FUNCTION_BLOCK Hexapod_Leg
VAR_INPUT
	Axis1, Axis2, Axis3	: Axis;
END_VAR
VAR_OUTPUT
END_VAR
VAR
	Axis_Leg		: ARRAY [1..3] OF Axis;
	Axis_Number		: INT;
	Axis_HomeDone	: ARRAY [1..3] OF BOOL;
	HomeDone		: BOOL;
END_VAR

Axis_Leg[1] := Axis1;
Axis_Leg[2] := Axis2;
Axis_Leg[3] := Axis3;

METHOD Home
VAR_INPUT
	Axis1_HomeSet	: BOOL;
	Axis2_HomeSet	: BOOL;
	Axis3_HomeSet	: BOOL;
END_VAR
VAR_OUTPUT	
END_VAR
VAR
	Axis_HomeSet	: BOOL;
END_VAR
IF Axis_HomeDone[1] AND Axis_HomeDone[2] AND Axis_HomeDone[2] THEN
	HomeDone := TRUE;
END_IF

Axis_HomeDone[1] := Axis1.State_HomeDone;
Axis_HomeDone[2] := Axis2.State_HomeDone;
Axis_HomeDone[3] := Axis3.State_HomeDone;
END_METHOD

PROPERTY State_HomeDone : BOOL
GET
State_HomeDone := HomeDone;
END_GET
END_PROPERTY

END_FUNCTION_BLOCK

(* stored: Version 1.1.0.1, ProductVersion 3.1.4020.12
   POU Hexapod_Leg: Id {49eba7d8-d2c8-4ac9-8090-16d605a814cb}, SpecialFunc None
   Method Home: Id {f793b9f5-69c0-4aee-af04-1fe207aaecb6}
   Property State_HomeDone: Id {8ca86c01-ddc8-4dc1-9d24-6379a91e4e8a}
   Get Get: Id {9a83aeec-779d-4e61-86ae-2b2c09c8cf87} *)
